(* CoDeSys 2.3 export: TYPETHERNET_BUFFER.EXP *)

(* Data type *)
TYPE typEthernet_BUFFER :
	STRUCT
		Index		:	INT;
		Data		:	ARRAY[1..1500] OF BYTE;
	END_STRUCT
END_TYPE
